# EPICS substitutions: epics-ioc-dev/reaktor/reaktorApp/Db/eurotherm24xx32xx.substitutions
file db/aiFloat64.template

{ pattern {X,           Y,            PORT,       OFFSET,   DATA_TYPE,     PREC,    SCAN}

{"$(P):$(R):", "$(N):iPV"	 ,       "$(I)",      1		,   INT16,         0,    "1 second"}
{"$(P):$(R):", "$(N):itSP"	 ,       "$(I)",      2		,   INT16,         0,    "1 second"}
{"$(P):$(R):", "$(N):itOP"	 ,       "$(I)",      3		,   INT16,         0,    "1 second"}
{"$(P):$(R):", "$(N):iW_SP"	 ,       "$(I)",      5		,   INT16,         0,    "1 second"}
{"$(P):$(R):", "$(N):irnGL"	 ,       "$(I)",      11	,   INT16,         0,    "1 second"}
{"$(P):$(R):", "$(N):irnGH"	 ,       "$(I)",      12	,   INT16,         0,    "1 second"}
{"$(P):$(R):", "$(N):iSP_1"	 ,       "$(I)",      24	,   INT16,         0,    "1 second"}
{"$(P):$(R):", "$(N):iSP_2"	 ,       "$(I)",      25	,   INT16,         0,    "1 second"}
{"$(P):$(R):", "$(N):iSbOP"	 ,       "$(I)",      34	,   INT16,         0,    "1 second"}
{"$(P):$(R):", "$(N):iSPrr"	 ,       "$(I)",      35	,   INT16,         0,    "1 second"}
{"$(P):$(R):", "$(N):iSP_H"	 ,       "$(I)",      111	,   INT16,         0,    "1 second"}
{"$(P):$(R):", "$(N):iSP_L"	 ,       "$(I)",      112	,   INT16,         0,    "1 second"}
{"$(P):$(R):", "$(N):iIM"	 ,       "$(I)",      199	,   INT16,         0,    "1 second"}
{"$(P):$(R):", "$(N):iCtrl"	 ,       "$(I)",      512	,   INT16,         0,    "1 second"}
{"$(P):$(R):", "$(N):iPwrF"	 ,       "$(I)",      518	,   INT16,         0,    "1 second"}
{"$(P):$(R):", "$(N):idEcP"	 ,       "$(I)",      525	,   INT16,         0,    "1 second"}
{"$(P):$(R):", "$(N):irmPU"	 ,       "$(I)",      531	,   INT16,         0,    "1 second"}
{"$(P):$(R):", "$(N):iinPT"	 ,       "$(I)",      12290	,   INT16,         0,    "1 second"}
{"$(P):$(R):", "$(N):iunit"	 ,       "$(I)",      516	,	INT16,         0,    "1 second"}
{"$(P):$(R):", "$(N):itune"	 ,       "$(I)",      270	,	INT16,         0,    "1 second"}
{"$(P):$(R):", "$(N):idrA"	 ,       "$(I)",      271	,	INT16,         0,    "1 second"}
{"$(P):$(R):", "$(N):idrAt"	 ,       "$(I)",      100	,	INT16,         0,    "1 second"}
{"$(P):$(R):", "$(N):iGSP"	 ,       "$(I)",      153	,	INT16,         0,    "1 second"}
{"$(P):$(R):", "$(N):iSET"	 ,       "$(I)",      72 	,	INT16,         0,    "1 second"}
{"$(P):$(R):", "$(N):iPbc"	 ,       "$(I)",      90 	,	INT16,         0,    "1 second"}
{"$(P):$(R):", "$(N):idbc"	 ,       "$(I)",      91 	,	INT16,         0,    "1 second"}
{"$(P):$(R):", "$(N):iFFPb"	 ,       "$(I)",      97 	,	INT16,         0,    "1 second"}
{"$(P):$(R):", "$(N):iFFtr"	 ,       "$(I)",      98 	,	INT16,         0,    "1 second"}
{"$(P):$(R):", "$(N):iFFdu"	 ,       "$(I)",      99 	,	INT16,         0,    "1 second"}
{"$(P):$(R):", "$(N):iPb"	 ,       "$(I)",      6  	,	INT16,         0,    "1 second"}
{"$(P):$(R):", "$(N):iti"	 ,       "$(I)",      8  	,	INT16,         0,    "1 second"}
{"$(P):$(R):", "$(N):itd"	 ,       "$(I)",      9  	,	INT16,         0,    "1 second"}
{"$(P):$(R):", "$(N):ires"	 ,       "$(I)",      28 	,	INT16,         0,    "1 second"}
{"$(P):$(R):", "$(N):iHcb"	 ,       "$(I)",      18 	,	INT16,         0,    "1 second"}
{"$(P):$(R):", "$(N):iLcb"	 ,       "$(I)",      17 	,	INT16,         0,    "1 second"}
{"$(P):$(R):", "$(N):irElc"	 ,       "$(I)",      19 	,	INT16,         0,    "1 second"}
{"$(P):$(R):", "$(N):iPb2"	 ,       "$(I)",      48  	,	INT16,         0,    "1 second"}
{"$(P):$(R):", "$(N):iti2"	 ,       "$(I)",      49 	,	INT16,         0,    "1 second"}
{"$(P):$(R):", "$(N):itd2"	 ,       "$(I)",      51  	,	INT16,         0,    "1 second"}
{"$(P):$(R):", "$(N):ires2"	 ,       "$(I)",      50 	,	INT16,         0,    "1 second"}
{"$(P):$(R):", "$(N):iHcb2"	 ,       "$(I)",      118 	,	INT16,         0,    "1 second"}
{"$(P):$(R):", "$(N):iLcb2"	 ,       "$(I)",      117 	,	INT16,         0,    "1 second"}
{"$(P):$(R):", "$(N):irEl2"	 ,       "$(I)",      52 	,	INT16,         0,    "1 second"}
{"$(P):$(R):", "$(N):iOPLo"	 ,       "$(I)",      31 	,	INT16,         0,    "1 second"}
{"$(P):$(R):", "$(N):iOPHi"	 ,       "$(I)",      30 	,	INT16,         0,    "1 second"}
#ALARM1
#{"$(P):$(R):", "$(N):iAL1Th" ,       "$(I)",      13 	,	INT16,         0,    "1 second"}
#{"$(P):$(R):", "$(N):iAL1Hy" ,       "$(I)",      47 	,	INT16,         0,    "1 second"}
#{"$(P):$(R):", "$(N):iAL1De" ,       "$(I)",      221 	,	INT16,         0,    "1 second"}
#{"$(P):$(R):", "$(N):iAL1Ty" ,       "$(I)",      10240,	INT16,         0,    "1 second"}
#{"$(P):$(R):", "$(N):iAL1Thr",       "$(I)",      10241,	INT16,         0,    "1 second"}
#{"$(P):$(R):", "$(N):iAL1Hys",       "$(I)",      10242,	INT16,         0,    "1 second"}
#{"$(P):$(R):", "$(N):iAL1Ref",       "$(I)",      10243,	INT16,         0,    "1 second"}
#{"$(P):$(R):", "$(N):iAL1Lat",       "$(I)",      10244,	INT16,         0,    "1 second"}
#{"$(P):$(R):", "$(N):iAL1Pri",       "$(I)",      10245,	INT16,         0,    "1 second"}
#{"$(P):$(R):", "$(N):iAL1Blo",       "$(I)",      10246,	INT16,         0,    "1 second"}
#{"$(P):$(R):", "$(N):iAL1Inh",       "$(I)",      10247,	INT16,         0,    "1 second"}
#{"$(P):$(R):", "$(N):iAL1Del",       "$(I)",      10248,	INT16,         0,    "1 second"}
#{"$(P):$(R):", "$(N):iAL1Out",       "$(I)",      10249,	INT16,         0,    "1 second"}
#{"$(P):$(R):", "$(N):iAL1Ack",       "$(I)",      10250,	INT16,         0,    "1 second"}
##ALARM GENERAL
#{"$(P):$(R):", "$(N):iALmSum",       "$(I)",      260	,	INT16,         0,    "1 second"}
#{"$(P):$(R):", "$(N):iALmAny",       "$(I)",      261	,	INT16,         0,    "1 second"}
}

file db/aoFloat64.template

{ pattern {X,           Y,            PORT,       OFFSET,DATA_TYPE, PREC,			EGU,  DESC,	  HOPR, LOPR}

# Control
{"$(P):$(R):", "$(N):otSP"	  ,       "$(O)",      2	,   INT16,     0,     "0.1degC",	"",   6000,  200}
{"$(P):$(R):", "$(N):oSPrr"	  ,       "$(O)",      35	,   INT16,     0, "0.1degC/min",	"",    100,    1}
{"$(P):$(R):", "$(N):oSP_H"	  ,       "$(O)",      111	,   INT16,     0,     "0.1degC",	"",   6000,  251}
{"$(P):$(R):", "$(N):oSP_L"	  ,       "$(O)",      112	,   INT16,     0,	  "0.1degC",	"",	   250,  200}
# Autotune
{"$(P):$(R):", "$(N):otune"	  ,       "$(O)",      270	,	INT16,     0,	         "",	"",		  ,	    }
{"$(P):$(R):", "$(N):odrA"	  ,       "$(O)",      271	,	INT16,     0,	         "",	"",		  ,	    }
{"$(P):$(R):", "$(N):odrAt"	  ,       "$(O)",      100	,	INT16,     0,	         "",	"",		  ,	    }
# PID
{"$(P):$(R):", "$(N):oGSP"	  ,       "$(O)",      153	,	INT16,     0,	         "",	"",		  ,	    }
{"$(P):$(R):", "$(N):oSET"	  ,       "$(O)",      72 	,	INT16,     0,	         "",	"",		  ,	    }
{"$(P):$(R):", "$(N):oFFPb"	  ,       "$(O)",      97 	,	INT16,     0,	         "",	"",		  ,	    }
{"$(P):$(R):", "$(N):oFFtr"	  ,       "$(O)",      98 	,	INT16,     0,	         "",	"",		  ,	    }
{"$(P):$(R):", "$(N):oFFdu"	  ,       "$(O)",      99 	,	INT16,     0,	         "",	"",		  ,	    }
{"$(P):$(R):", "$(N):oPb"	  ,       "$(O)",      6  	,	INT16,     0,	         "",	"",		  ,	    }
{"$(P):$(R):", "$(N):oti"	  ,       "$(O)",      8  	,	INT16,     0,	         "",	"",		  ,	    }
{"$(P):$(R):", "$(N):otd"	  ,       "$(O)",      9  	,	INT16,     0,	         "",	"",		  ,	    }
{"$(P):$(R):", "$(N):ores"	  ,       "$(O)",      28 	,	INT16,     0,	         "",	"",		  ,	    }
{"$(P):$(R):", "$(N):oHcb"	  ,       "$(O)",      18 	,	INT16,     0,	         "",	"",		  ,	    }
{"$(P):$(R):", "$(N):oLcb"	  ,       "$(O)",      17 	,	INT16,     0,	         "",	"",		  ,	    }
{"$(P):$(R):", "$(N):oPb2"	  ,       "$(O)",      48  	,	INT16,     0,	         "",	"",		  ,	    }
{"$(P):$(R):", "$(N):oti2"	  ,       "$(O)",      49 	,	INT16,     0,	         "",	"",		  ,	    }
{"$(P):$(R):", "$(N):otd2"	  ,       "$(O)",      51  	,	INT16,     0,	         "",	"",		  ,	    }
{"$(P):$(R):", "$(N):ores2"	  ,       "$(O)",      50 	,	INT16,     0,	         "",	"",		  ,	    }
{"$(P):$(R):", "$(N):oHcb2"	  ,       "$(O)",      118 	,	INT16,     0,	         "",	"",		  ,	    }
{"$(P):$(R):", "$(N):oLcb2"	  ,       "$(O)",      117 	,	INT16,     0,	         "",	"",		  ,	    }
# PID (Cooling Options)
#{"$(P):$(R):", "$(N):oPbc"	 ,       "$(O)",      90 	,	INT16,     0,	         "",	"",		  ,	    }
#{"$(P):$(R):", "$(N):odbc"	 ,       "$(O)",      91 	,	INT16,     0,	         "",	"",		  ,	    }
#{"$(P):$(R):", "$(N):orElc" ,       "$(O)",      19 	,	INT16,     0,	         "",	"",		  ,	    }
#{"$(P):$(R):", "$(N):orEl2" ,       "$(O)",      52 	,	INT16,     0,	         "",	"",		  ,	    }
# Outputlevel
{"$(P):$(R):", "$(N):oOPLo"  ,       "$(O)",      31	,	INT16,     0,	     "0.1%",	"",	  1000,	   0}
{"$(P):$(R):", "$(N):oOPHi"  ,       "$(O)",      30	,	INT16,     0,	     "0.1%",	"",	  1000,	   0}
# Configuration Menue/Mode: Attention! Restart after switching back to normal mode!
{"$(P):$(R):", "$(N):oIM"	 ,       "$(O)",      199	,   INT16,     0,            "",	"",	     2,	   0}
{"$(P):$(R):", "$(N):ounit"	 ,       "$(O)",      516	,	INT16,     0, 			 "",	"",	     3,	   0}
{"$(P):$(R):", "$(N):ormPU"	 ,       "$(O)",      531	,   INT16,     0, 			 "",	"",	     2,	   0}
{"$(P):$(R):", "$(N):odEcP"	 ,       "$(O)",      525	,   INT16,     0, 			 "",	"",	     2,	   0}
{"$(P):$(R):", "$(N):ornGL"	 ,       "$(O)",      11	,   INT16,     0,     "0.1degC",	"",    200,  200}
{"$(P):$(R):", "$(N):ornGH"	 ,       "$(O)",      12	,   INT16,     0,     "0.1degC",	"",   6000, 6000}
{"$(P):$(R):", "$(N):oSP_1"	 ,       "$(O)",      24	,   INT16,     0,     "0.1degC",	"",   6000,  200}
{"$(P):$(R):", "$(N):oSP_2"	 ,       "$(O)",      25	,   INT16,     0,     "0.1degC",	"",    250,  200}
{"$(P):$(R):", "$(N):oCtrl"	 ,       "$(O)",      512	,   INT16,     0,            "",	"",	     4,	   0}
{"$(P):$(R):", "$(N):oPwrF"	 ,       "$(O)",      518	,   INT16,     0, 	  		 "",	"",	     2,	   0}
{"$(P):$(R):", "$(N):oinPT"	 ,       "$(O)",      12290	,   INT16,     0, 	  		 "",	"",	     1,	   1}
##ALARM1
#{"$(P):$(R):", "$(N):oAL1Th" ,       "$(O)",      13 	,	INT16,     0,            "",    "",       ,     }
#{"$(P):$(R):", "$(N):oAL1Hy" ,       "$(O)",      47 	,	INT16,     0,            "",    "",       ,     }
#{"$(P):$(R):", "$(N):oAL1De" ,       "$(O)",      221 	,	INT16,     0,            "",    "",       ,     }
#{"$(P):$(R):", "$(N):oAL1Ty" ,       "$(O)",      10240,	INT16,     0,            "",    "",       ,     }
#{"$(P):$(R):", "$(N):oAL1Thr",       "$(O)",      10241,	INT16,     0,            "",    "",       ,     }
#{"$(P):$(R):", "$(N):oAL1Hys",       "$(O)",      10242,	INT16,     0,            "",    "",       ,     }
#{"$(P):$(R):", "$(N):oAL1Ref",       "$(O)",      10243,	INT16,     0,            "",    "",       ,     }
#{"$(P):$(R):", "$(N):oAL1Lat",       "$(O)",      10244,	INT16,     0,            "",    "",       ,     }
#{"$(P):$(R):", "$(N):oAL1Pri",       "$(O)",      10245,	INT16,     0,            "",    "",       ,     }
#{"$(P):$(R):", "$(N):oAL1Blo",       "$(O)",      10246,	INT16,     0,            "",    "",       ,     }
#{"$(P):$(R):", "$(N):oAL1Inh",       "$(O)",      10247,	INT16,     0,            "",    "",       ,     }
#{"$(P):$(R):", "$(N):oAL1Del",       "$(O)",      10248,	INT16,     0,            "",    "",       ,     }
#{"$(P):$(R):", "$(N):oAL1Out",       "$(O)",      10249,	INT16,     0,            "",    "",       ,     }
#{"$(P):$(R):", "$(N):oAL1Ack",       "$(O)",      10250,	INT16,     0,            "",    "",       ,     }
}
